// TIA Portal V21 export
VAR_GLOBAL   // PLC tag table "K_TipoMotore"
END_VAR
VAR_GLOBAL CONSTANT   // user constants
   K_TipoMotore_Teleruttore1Dir : Int := 0;
   K_TipoMotore_Teleruttore2Dir : Int := 1;
   K_TipoMotore_InverterMitsubishi : Int := 2;
   K_TipoMotore_InverterSiemens : Int := 3;
   K_TipoMotore_InverterSchneider : Int := 4;
   K_TipoMotore_InverterMovimot : Int := 5;
   K_TipoMotore_InverterMoviGear : Int := 6;
   K_TipoMotore_InverterDanfoss : Int := 7;
   K_TipoMotore_InverterMovitrac : Int := 8;
   K_TipoMotore_InverterINVT : Int := 9;
   K_TipoMotore_InverterNIDEC : Int := 10;
   K_TipoMotore_InverterKEB : Int := 11;
   "K_TipoMotore_AzionamentoFesto_CMMT-ST" : Int := 12;
END_VAR
